
(* ===== HMI "HiddenHmiRTDeviceFaceplateTypes" =====

HMI tags "9ca7d841-4e4d-4293-b7f5-7bf308eb5ab1"
   "ExtProg" : 3501ddcb-ead9-49b1-ad45-e1bdd97be0cf, internal
*)

(* ===== HMI "HMI_RT_1" =====

HMI tags "WinProgManager"
   "_WINPROGMANAGER_" : 3501ddcb-ead9-49b1-ad45-e1bdd97be0cf, internal
*)